TYPE ST_AlarmEntry :
STRUCT
    pAlarm : POINTER TO ST_Alarm;     
    sName : STRING(50);               
END_STRUCT
END_TYPE

(* stored: Version 1.1.0.1, ProductVersion 3.1.4026.11
   DUT ST_AlarmEntry: Id {ace690c2-6328-4f6e-b841-e69cd57e66ab} *)
